PROGRAM LLD
VAR
	count : INT := 0;
	reset : BOOL := FALSE;
	
END_VAR
VAR // added by the converter: edge detectors and wires of the graphical bodies
    _w1, _w2 : BOOL;
END_VAR

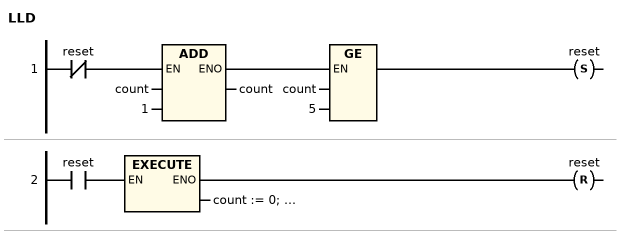
// NETWORK 1
_w1 := NOT reset;
IF _w1 THEN count := count + 1; END_IF
reset S= _w1 AND count >= 5;

// NETWORK 2
_w2 := reset;
IF _w2 THEN count := 0; END_IF
reset R= _w2;

END_PROGRAM

(* stored: Version 1.1.0.1, ProductVersion 3.1.4024.12
   POU LLD: Id {fd6a5808-02df-4a61-921b-ef422415d1b4}, SpecialFunc None *)
